FUNCTION_BLOCK AGENT_SERVER (* Service Interface Function Block Type *)
  (* Standard: 61499-2; Description: This Service Interface Function Block listens for in-coming connection requests from the remote diagnostic agent. Each packet received carries a data value that is to be output to the function block that is being tested. *)
  (* Version 1.0, 2019-01-10, badger *)
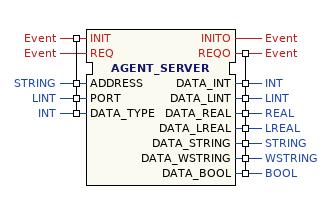
  EVENT_INPUT
    INIT WITH ADDRESS, PORT, DATA_TYPE; (* Service Initialization *)
    REQ; (* Service Request *)
  END_EVENT
  EVENT_OUTPUT
    INITO; (* Used to trigger the initialisation of other diagnostic AGENT_SEND function blocks that are being used to assist with the diagnosis. *)
    REQO WITH DATA_INT, DATA_LINT, DATA_REAL, DATA_LREAL, DATA_STRING, DATA_WSTRING, DATA_BOOL; (* Used to alert the function block that is being tested that new data is available on the agreed output. *)
  END_EVENT
  VAR_INPUT
    ADDRESS : STRING; (* Address that this agent function block is listening on for incoming connection requests. *)
    PORT : LINT; (* Port that this function block is listening on. *)
    DATA_TYPE : INT; (* Enumerated data type used to determine what type of data should be output from this function block. *)
  END_VAR
  VAR_OUTPUT
    DATA_INT : INT; (* Integer data type *)
    DATA_LINT : LINT; (* Long integer data type. *)
    DATA_REAL : REAL; (* Real data type *)
    DATA_LREAL : LREAL; (* Long Real data type *)
    DATA_STRING : STRING; (* String data type *)
    DATA_WSTRING : WSTRING; (* Wide String data type. *)
    DATA_BOOL : BOOL; (* Boolean data type. *)
  END_VAR
  SERVICE APPLICATION/RESOURCE (* Service Interface Function Block Type *)
    SEQUENCE normal_establishment
      APPLICATION.INIT+(PARAMS) -> RESOURCE.initialize(PARAMS) -> APPLICATION.INITO+();
    END_SEQUENCE
    SEQUENCE unsuccessful_establishment
      APPLICATION.INIT+(PARAMS) -> RESOURCE.initialize(PARAMS) -> APPLICATION.INITO-(STATUS);
    END_SEQUENCE
    SEQUENCE request_confirm
      APPLICATION.REQ+(SD) -> RESOURCE.request(SD) -> APPLICATION.CNF+(RD);
    END_SEQUENCE
    SEQUENCE request_inhibited
      APPLICATION.REQ-(SD) -> APPLICATION.CNF-(STATUS);
    END_SEQUENCE
    SEQUENCE request_error
      APPLICATION.REQ+(SD) -> RESOURCE.request(SD) -> APPLICATION.CNF-(STATUS);
    END_SEQUENCE
    SEQUENCE indication_response
      RESOURCE.indicate(RD) -> APPLICATION.IND+(RD);
      APPLICATION.RSP(QI,SD) -> RESOURCE.response(QI,SD);
    END_SEQUENCE
    SEQUENCE indication_inhibited
      RESOURCE.indicate(RD,QI=FALSE) -> RESOURCE.inhibited();
    END_SEQUENCE
    SEQUENCE error_indication
      RESOURCE.error(STATUS) -> APPLICATION.IND-(STATUS);
    END_SEQUENCE
    SEQUENCE application_initiated_termination
      APPLICATION.INIT-() -> RESOURCE.terminate() -> APPLICATION.INITO-(STATUS);
    END_SEQUENCE
    SEQUENCE resource_initiated_termination
      -> APPLICATION.INITO-(STATUS);
    END_SEQUENCE
  END_SERVICE
END_FUNCTION_BLOCK
